// TIA Portal V17 export
// export: Created 2024-06-14T09:53:52.3124871Z, ExportSetting WithDefaults, DisplayName Totally Integrated Automation Portal, DisplayVersion V17, DisplayName TIA Portal Openness, DisplayVersion V17, DisplayName TIA Portal Version Control Interface, DisplayVersion V17, DisplayName Simotion SCOUT TIA, DisplayVersion 5.4.3.0, DisplayName SINAMICS Startdrive Advanced, DisplayVersion V17 SP1 Update 1, DisplayName SINAMICS Startdrive G110M, G120, G120C, G120D, G120P, G115D, DisplayVersion V17 SP1 Update 1, DisplayName SINAMICS Startdrive G130, G150, S120, S150, SINAMICS MV, S210, DisplayVersion V17 SP1 Update 1, DisplayName STEP 7 Professional, DisplayVersion V17, DisplayName STEP 7 Safety, DisplayVersion V17, DisplayName WinCC Professional, DisplayVersion V17
TYPE "Mod_Client_Data"
// stored: IsFailsafeCompliant false
   STRUCT
      request : Bool;
      enable : Bool;
      disconnect : Bool;
      done : Bool;
      busy : Bool;
      error : Bool;
      status : Word;
      statusSave : Word;
      modbusMode : USInt;
      modbusDataAddress : UDInt;
      modbusDataLen : UInt;
   END_STRUCT;
END_TYPE
